{attribute addProperty BoxType "EP2339-0003-0016"}
{attribute addProperty Id "DI_Inputs_ChannelAT %I*ARRAY[0..11] OF DI_Inputs_Channel_595007DD176220DO_Outputs_ChannelAT %Q*ARRAY[0..8] OF DO_Outputs_Channel_33B76376128160WcStateAT %I*WcState_98A4DF7520.250InfoDataAT %I*InfoData_BC63D37F80100"}
{attribute addProperty CRC "1382427570"}
{attribute addProperty SizeInBites "386"}
{attribute addProperty SizeInBytes "48.25"}
TYPE EP2339_41D05C24 :
STRUCT
	{attribute addProperty Name "DI_Inputs_Channel"}
	DI_Inputs_Channel : ARRAY[0..11] OF DI_Inputs_Channel_595007DD;
	{attribute addProperty Name "DO_Outputs_Channel"}
	DO_Outputs_Channel : ARRAY[0..8] OF DO_Outputs_Channel_33B76376;
	{attribute addProperty Name "WcState"}
	WcState : WcState_98A4DF75;
	{attribute addProperty Name "InfoData"}
	InfoData : InfoData_BC63D37F;
END_STRUCT
END_TYPE

(* stored: Version 1.2.0.0, ProductVersion 3.1.4024.9
   DUT EP2339_41D05C24: Id {f3756cff-042d-45ed-a963-a0d77973174c} *)
